(* PLC project Unnamed, Unknown Unnamed 1 *)
(* stored: creationDateTime 2025-12-22T17:40:39, modificationDateTime 2025-12-28T10:44:06 *)

PROGRAM program0
  VAR
    LocalVar0 : DINT;
    LocalVar1 : DINT;
  END_VAR

            LocalVar0 := LocalVar1;

          
END_PROGRAM

CONFIGURATION config
  RESOURCE resource1 ON PLC
    TASK task0(INTERVAL := T#20ms, PRIORITY := 0);
    PROGRAM instance0 WITH task0 : program0;
  END_RESOURCE
END_CONFIGURATION
